FUNCTION_BLOCK hundredMStoS (* A simple FB with a single algorithm and REQ/CNF pair *)
  (* Standard: 61499-1 *)
  (* Version 0.0, 2006-09-03, JHC, Holobloc Inc *)
  (* Compiler header: package fb.rt.student; *)
  (* Compiler classdef: SimpleFB *)
  (* Compiler Java Sun JDK 1.5.0 *)
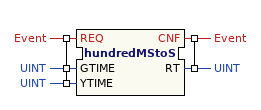
  EVENT_INPUT
    REQ WITH GTIME, YTIME; (* Normal Execution Request *)
  END_EVENT
  EVENT_OUTPUT
    CNF WITH RT; (* Execution Confirmation *)
  END_EVENT
  VAR_INPUT
    GTIME : UINT;
    YTIME : UINT;
  END_VAR
  VAR_OUTPUT
    RT : UINT;
  END_VAR
  ALGORITHM REQ IN ST: (* Normally executed algorithm *)
IF GTIME>=10 THEN
RT := ((GTIME - 1 - ((GTIME - 1) MOD 10))/10) + 1;
ELSIF (GTIME<10 AND GTIME>0) THEN
RT := 1;
ELSIF (GTIME=0 AND YTIME>=10) THEN
RT := ((YTIME - 1 - ((YTIME - 1) MOD 10))/10) + 1;
ELSIF (GTIME=0 AND YTIME<10 AND YTIME>0) THEN
RT := 1;
ELSE
RT := 0;
END_IF;
  END_ALGORITHM
END_FUNCTION_BLOCK
